PROGRAM MAIN
VAR
END_VAR

END_PROGRAM

(* stored: Version 1.1.0.1
   POU MAIN: Id {b69c4433-8053-4e54-b9ef-a688e047d957} *)
